FUNCTION_BLOCK LinksRechts (* Basic FB with Links-Rechts *)
  (* Standard: 61499-2; Description: Copyright (c) 2025 HR Agrartechnik GmbH This program and the accompanying materials are made available under the terms of the Eclipse Public License 2.0 which is available at https://www.eclipse.org/legal/epl-2.0/ SPDX-License-Identifier: EPL-2.0 Nur Rechtslauf ist vorrangig vor Nur Linkslauf. *)
  (* Version 1.0, 2025-05-23, Franz Höpfinger, HR Agrartechnik GmbH *)
  PACKAGE logiBUS::utils::sequence::verteiler;
  IMPORT Verteiler::LinksRechts::STATES;
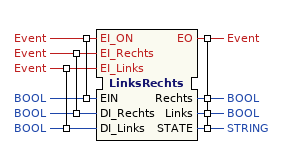
  EVENT_INPUT
    EI_ON WITH EIN; (* Einschalten *)
    EI_Rechts WITH DI_Rechts;
    EI_Links WITH DI_Links;
  END_EVENT
  EVENT_OUTPUT
    EO WITH Rechts, Links, STATE;
  END_EVENT
  VAR_INPUT
    EIN : BOOL; (* Einschalten *)
    DI_Rechts : BOOL; (* Nur Rechtslauf *)
    DI_Links : BOOL; (* Nur Linkslauf *)
  END_VAR
  VAR_OUTPUT
    Rechts : BOOL; (* Rechtslauf *)
    Links : BOOL; (* Linkslauf *)
    STATE : STRING;
  END_VAR
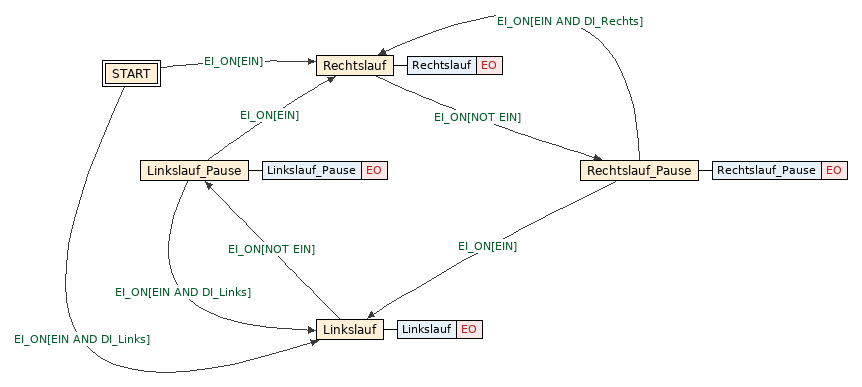
  EC_STATES
    START; (* Initial State *)
    Rechtslauf : Rechtslauf -> EO;
    Rechtslauf_Pause : Rechtslauf_Pause -> EO;
    Linkslauf : Linkslauf -> EO;
    Linkslauf_Pause : Linkslauf_Pause -> EO;
  END_STATES
  EC_TRANSITIONS
    START TO Linkslauf := EI_ON[EIN AND DI_Links];
    START TO Rechtslauf := EI_ON[EIN];
    Rechtslauf TO Rechtslauf_Pause := EI_ON[NOT EIN];
    Rechtslauf_Pause TO Rechtslauf := EI_ON[EIN AND DI_Rechts];
    Rechtslauf_Pause TO Linkslauf := EI_ON[EIN];
    Linkslauf TO Linkslauf_Pause := EI_ON[NOT EIN];
    Linkslauf_Pause TO Linkslauf := EI_ON[EIN AND DI_Links];
    Linkslauf_Pause TO Rechtslauf := EI_ON[EIN];
  END_TRANSITIONS
  ALGORITHM Rechtslauf IN ST:
Rechts := BOOL#TRUE;
Links := BOOL#FALSE;
STATE := STATES::Rechtslauf;
  END_ALGORITHM
  ALGORITHM Linkslauf IN ST:
Rechts := BOOL#FALSE;
Links := BOOL#TRUE;
STATE := STATES::Linkslauf;
  END_ALGORITHM
  ALGORITHM Linkslauf_Pause IN ST:
Rechts := BOOL#FALSE;
Links := BOOL#FALSE;
STATE := STATES::Linkslauf_Pause;
  END_ALGORITHM
  ALGORITHM Rechtslauf_Pause IN ST:
Rechts := BOOL#FALSE;
Links := BOOL#FALSE;
STATE := STATES::Rechtslauf_Pause;
  END_ALGORITHM
END_FUNCTION_BLOCK
